///EL1809 | HD EtherCAT Terminals, 16-channel digital input 24 V DC, 3 ms
FUNCTION_BLOCK EL1809

VAR_INPUT
    En              : BOOL;
    iTerminal_ID    : INT;
    ErrorSystem     : POINTER TO ST_ErrorSystem;
END_VAR

VAR_OUTPUT
    EnO                 : BOOL;
    bError              : BOOL;
	sErrorMessage       : STRING;
	bBI_1                AT %I*  : BOOL:=FALSE;
	bBI_2                AT %I*  : BOOL:=FALSE;
	bBI_3                AT %I*  : BOOL:=FALSE;
	bBI_4                AT %I*  : BOOL:=FALSE;
	bBI_5                AT %I*  : BOOL:=FALSE;
	bBI_6                AT %I*  : BOOL:=FALSE;
	bBI_7                AT %I*  : BOOL:=FALSE;
	bBI_8                AT %I*  : BOOL:=FALSE;
	bBI_9                AT %I*  : BOOL:=FALSE;
	bBI_10               AT %I*  : BOOL:=FALSE;
	bBI_11               AT %I*  : BOOL:=FALSE;
	bBI_12               AT %I*  : BOOL:=FALSE;
	bBI_13               AT %I*  : BOOL:=FALSE;
	bBI_14               AT %I*  : BOOL:=FALSE;
	bBI_15               AT %I*  : BOOL:=FALSE;
	bBI_16               AT %I*  : BOOL:=FALSE;
END_VAR

VAR
    WcState_WcState     AT %I*  : BOOL := TRUE;  // invalid
    InfoData_State      AT %I*  : UINT := 0;
    //dBI_all                     : INT  := 0;
    //FB-s
    EL1809_Error      : FB_TerminalError;
END_VAR

(*
* TODO: DONE!
*)
EnO:=En;
(*dBI_all.0:=bBI_1;
dBI_all.1:=bBI_2;
dBI_all.2:=bBI_3;
dBI_all.3:=bBI_4;
dBI_all.4:=bBI_5;
dBI_all.5:=bBI_6;
dBI_all.6:=bBI_7;
dBI_all.7:=bBI_8;
dBI_all.8:=bBI_9;
dBI_all.9:=bBI_10;
dBI_all.10:=bBI_11;
dBI_all.11:=bBI_12;
dBI_all.12:=bBI_13;
dBI_all.13:=bBI_14;
dBI_all.14:=bBI_15;
dBI_all.15:=bBI_16;*)

//Error FB instance
EL1809_Error(
    En                  := TRUE,
    iTerminal_ID        := iTerminal_ID,
    bWcState            := WcState_WcState,
    uiInfoData_State    := InfoData_State,
    pErrorSystem        := ErrorSystem,
    bError              => bError,
);

IF bError THEN
	sErrorMessage:=EL1809_Error.ErrorData.sErrorMessage;
ELSE
	sErrorMessage:='';
END_IF

END_FUNCTION_BLOCK

(* stored: Version 1.1.0.1, ProductVersion 3.1.4024.6
   POU EL1809: Id {1a348214-209a-44e9-9088-e1b46b9010e2}, SpecialFunc None *)
